// TIA Portal project "Curso PLC - Proyecto 1" (V17)

(* hardware
DEVICE "S7-1200 station_1"  S7-1200 Station
   slot 0: "Rack_0"  S7-1200 Rack  Rack  V1.0
   slot 1: "PLC_1"  CPU 1215C DC/DC/Rly  6ES7 215-1HG40-0XB0  V4.5
   slot 2: "DI 8x24VDC_1"  6ES7 221-1BF32-0XB0  V2.0
   slot 3: "DQ 8x24VDC _1"  SM 1222 DQ8 x 24VDC  6ES7 222-1BF32-0XB0  V2.0
*)

// ===== PLC "PLC_1"  CPU 1215C DC/DC/Rly =====

VAR_GLOBAL   // PLC tag table "Tabla de variables estándar"
   "PulsMarcha" AT %I0.0 : Bool;   // Pulsador de Marcha para Motor 1
   "ContMot" AT %Q0.0 : Bool;   // Salida de marcha motor 1
END_VAR

DATA_BLOCK "DB_GENERAL"   // DB1
{ S7_Optimized_Access := 'TRUE' }
VERSION : 0.1
   VAR
      EJEMPLO_BOOL : Bool;
      EJEMPLO_BYTE : Byte;
      EJEMPLO_WORD : Word;
      EJEMPLO_ENTERO : Int;
      EJEMPLO_DWORD : DWord;
      EJEMPLO_REAL : Real;
      EJEMPLO_CHAR : Char;
   END_VAR
BEGIN
END_DATA_BLOCK

ORGANIZATION_BLOCK "Main"   // OB1, LAD, ProgramCycle
TITLE = "Main Program Sweep (Cycle)"
{ S7_Optimized_Access := 'TRUE' }
VERSION : 0.1
   VAR_INPUT
      Initial_Call : Bool;   // Initial call of this OB
      Remanence : Bool;   // =True, if remanent data are available
   END_VAR
BEGIN

REGION Network 1: Salida de marcha motor 1
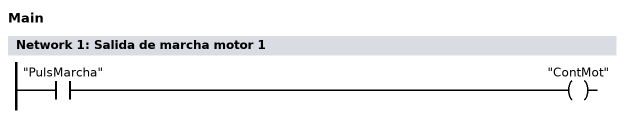
   RUNG wire#powerrail
      Contact( "PulsMarcha" )
      Coil( "ContMot" )
   END_RUNG
   // the same network as SCL:
   "ContMot" := "PulsMarcha";
END_REGION
END_ORGANIZATION_BLOCK